(*

.. <legal notes>

legal notes
=================
| SPDX-FileCopyrightText: © 2025 Oleksandr Tiutyk <trofimich@gmail.com>
| SPDX-License-Identifier: LGPL-3.0-only
| For details check: LGPL-3.0-only_

.. _LGPL-3.0-only: https://www.gnu.org/licenses/lgpl-3.0.en.html

.. </legal notes>

*)

PROGRAM SystemAnyTypeFactory
VAR
	_ClassName : STRING := __POUNAME();
END_VAR

{attribute 'monitoring' := 'call'}
PROPERTY ClassName : STRING
GET
ClassName := _ClassName;
END_GET
END_PROPERTY

METHOD CreateAnyTypeByAny : __SYSTEM.AnyType
VAR_INPUT
	anyValue : ANY;
END_VAR
CreateAnyTypeByAny := anyValue;
END_METHOD

METHOD CreateAnyTypeByGenericValue : __SYSTEM.AnyType
VAR_IN_OUT CONSTANT
	genericValue : GENERIC_VALUE;
END_VAR
CreateAnyTypeByGenericValue.TypeClass := SystemTypeClassConvertor.GetSystemTypeClassByDataType(genericValue.DataType);
CreateAnyTypeByGenericValue.pValue := genericValue.Address;
CreateAnyTypeByGenericValue.diSize := TO_DINT(genericValue.Size);
END_METHOD

END_PROGRAM

(* stored: Version 1.1.0.1
   POU SystemAnyTypeFactory: Id {2f1d6367-865e-4816-ae65-fc891ffa8aef}, SpecialFunc None
   Property ClassName: Id {a18dc19b-2cc2-4385-b86b-66fb39894a76}
   Get Get: Id {a9a7ad10-1195-4121-9ce8-7045b5415930}
   Method CreateAnyTypeByAny: Id {1f2becd5-4a43-4d75-827f-7c56c084215c}
   Method CreateAnyTypeByGenericValue: Id {73f9d3c1-a03b-4864-9d65-f396047544c5} *)
